{attribute 'qualified only'}
TYPE ENUM_Si_B4C_Coating_States :
(
	Unknown := 0,
    Si := 1,
    B4C := 2
);
END_TYPE

(* stored: Version 1.1.0.1, ProductVersion 3.1.4022.18
   DUT ENUM_Si_B4C_Coating_States: Id {05cb8cdb-5c23-4ac8-8acb-4957d82ceecd} *)
